{attribute addProperty BoxType "EK1101-0000-0016"}
{attribute addProperty Id "IDAT %I*UINT162"}
{attribute addProperty CRC "2432610056"}
{attribute addProperty SizeInBites "16"}
{attribute addProperty SizeInBytes "2"}
TYPE ID_90FEAF08 :
STRUCT
	{attribute addProperty Name "ID"}
	ID AT %I* : UINT;
END_STRUCT
END_TYPE

(* stored: Version 1.2.0.0, ProductVersion 3.1.4024.9
   DUT ID_90FEAF08: Id {4ca7b6c9-6036-4d0b-99fd-b8f60c90975a} *)
